{attribute 'qualified_only'}
{attribute 'strict'}
{attribute 'to_string'}
TYPE E_SeqDockingInterface :
(
	IDLE := 0,
	START := 1,
	
	OPEN_ALL_DOCKING_CLAMPS,
	
	CLOSE_ALL_DOCKING_CLAMPS,
	COMPRESS_ALL_SEAL,
	
	CLOSE_LOWER_DOCKING_CLAMPS,
	COMPRESS_LOWER_SEAL,
	CLOSE_UPPER_DOCKING_CLAMPS,
	COMPRESS_UPPER_SEAL,
	
	TB_DOCKED,
	CLOSE_DOOR_OPENER_RELEASING_PINS,
	CLOSE_DOOR_SHUTTER_RELEASING_PINS,
	RELEASE_UNLOCKING_PINS,
	OPEN_DOOR_SHUTTER,
	OPEN_DOOR_OPENER,
	
	INNER_DOOR_OPENED,
	CLOSE_DOOR_OPENER,
	CLOSE_DOOR_SHUTTER,
	LOCK_UNLOCKING_PINS,
	OPEN_DOOR_SHUTTER_2,
	
	READY := 10000,
	ERROR := 20000	
);
END_TYPE

(* stored: Version 1.1.0.1, ProductVersion 3.1.4024.12
   DUT E_SeqDockingInterface: Id {7699f56e-cf50-4a81-b35f-f3ec800bd102} *)
